FUNCTION_BLOCK FB_RS (* Bistable Function Block (reset dominant) *)
  (* Standard: 61131-3; Classification: bistable function block *)
  (* Version 1.0, 2009-09-14, 4DIAC-IDE, 4DIAC-Consortium *)
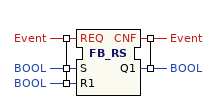
  EVENT_INPUT
    REQ WITH S, R1; (* Service Request *)
  END_EVENT
  EVENT_OUTPUT
    CNF WITH Q1; (* Confirmation of Requested Service *)
  END_EVENT
  VAR_INPUT
    S : BOOL; (* Set *)
    R1 : BOOL; (* Reset *)
  END_VAR
  VAR_OUTPUT
    Q1 : BOOL; (* Output *)
  END_VAR
  (* Service APPLICATION/RESOURCE: Bistable Function Block (reset dominant) *)
END_FUNCTION_BLOCK
